FUNCTION_BLOCK PUBLIC reset_errors
VAR
	 bStart          : BOOL := TRUE;
	 fbTimer         : TON;
	 fbTrigger       : R_TRIG;
	 tTimerValue     : TIME := T#1S;
END_VAR

GVL.robotdata.motorCword[0]:=128;
GVL.robotdata.motorCword[1]:=128;
GVL.robotdata.motorCword[2]:=128;
GVL.robotdata.motorCword[3]:=128;
fbTimer(IN := bStart, PT := tTimerValue);
motion_index:=max_location;
robotdata.motion_status:=MOTION_ENDED;
Locomotion_1_target_velocity:=0;
Locomotion_2_target_velocity:=0;

st_command.command:=0;

END_FUNCTION_BLOCK

(* stored: Version 1.1.0.1, ProductVersion 3.1.4024.12
   POU reset_errors: Id {7618a898-199c-40c8-b33c-864350276044}, SpecialFunc None *)
